// TIA Portal V17 export
// export: Created 2023-12-05T13:40:23.7935215Z, ExportSetting WithDefaults, DisplayName Totally Integrated Automation Portal, DisplayVersion V17, DisplayName TIA Portal Openness, DisplayVersion V17, DisplayName TIA Portal Version Control Interface, DisplayVersion V17, DisplayName SINAMICS Startdrive Advanced, DisplayVersion V17, DisplayName SINAMICS Startdrive G130, G150, S120, S150, SINAMICS MV, S210, DisplayVersion V17, DisplayName SINAMICS Startdrive G110M, G120, G120C, G120D, G120P, G115D, DisplayVersion V17, DisplayName STEP 7 Professional, DisplayVersion V17, DisplayName STEP 7 Safety, DisplayVersion V17, DisplayName WinCC Professional, DisplayVersion V17
FUNCTION "KNIFE_AND_SLUG_COUNTER_MANAGE" : Void   // FC402, LAD
{ S7_Optimized_Access := 'TRUE' }
VERSION : 0.1
// stored: AutoNumber false, IsIECCheckEnabled false, SetENOAutomatically false, UDAEnableTagReadback false
   VAR_TEMP   // added for the SCL form of the ladder/FBD networks
      _w1 : Bool;
      _w2 : Bool;
   END_VAR
BEGIN

REGION Network 1: -------------------------------------------------- KNIFE COUNTERS --------------------------------------------------
END_REGION

REGION Network 2: ST1OP02
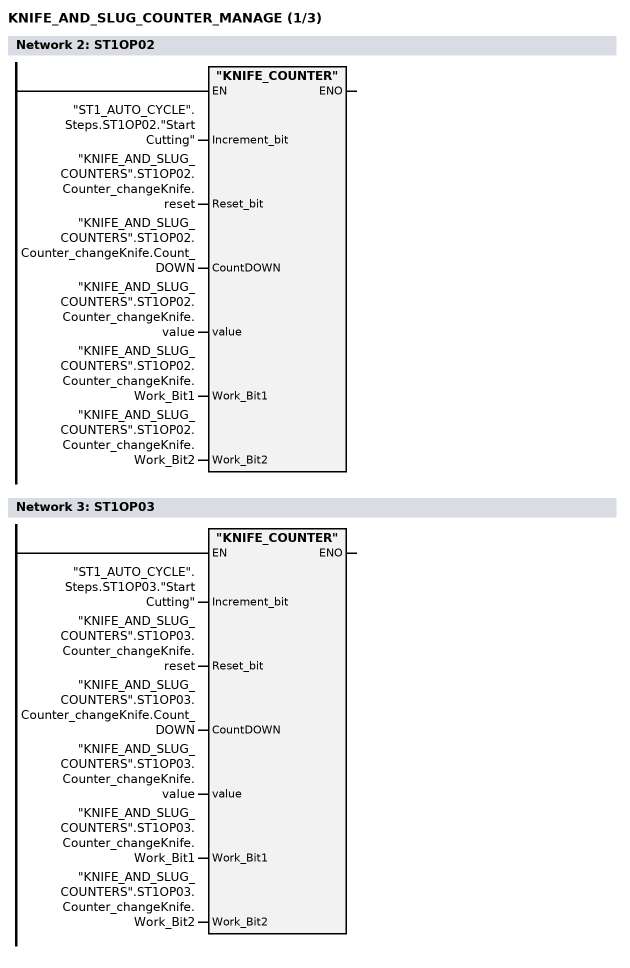
   RUNG wire#powerrail
      "KNIFE_COUNTER"(Increment_bit := "ST1_AUTO_CYCLE".Steps.ST1OP02."Start Cutting", Reset_bit := "KNIFE_AND_SLUG_COUNTERS".ST1OP02.Counter_changeKnife.reset, CountDOWN := "KNIFE_AND_SLUG_COUNTERS".ST1OP02.Counter_changeKnife.Count_DOWN, value := "KNIFE_AND_SLUG_COUNTERS".ST1OP02.Counter_changeKnife.value, Work_Bit1 := "KNIFE_AND_SLUG_COUNTERS".ST1OP02.Counter_changeKnife.Work_Bit1, Work_Bit2 := "KNIFE_AND_SLUG_COUNTERS".ST1OP02.Counter_changeKnife.Work_Bit2)
   END_RUNG
   // the same network as SCL:
   "KNIFE_COUNTER"(Increment_bit := "ST1_AUTO_CYCLE".Steps.ST1OP02."Start Cutting",
                   Reset_bit := "KNIFE_AND_SLUG_COUNTERS".ST1OP02.Counter_changeKnife.reset,
                   CountDOWN := "KNIFE_AND_SLUG_COUNTERS".ST1OP02.Counter_changeKnife.Count_DOWN,
                   value := "KNIFE_AND_SLUG_COUNTERS".ST1OP02.Counter_changeKnife.value,
                   Work_Bit1 := "KNIFE_AND_SLUG_COUNTERS".ST1OP02.Counter_changeKnife.Work_Bit1,
                   Work_Bit2 := "KNIFE_AND_SLUG_COUNTERS".ST1OP02.Counter_changeKnife.Work_Bit2);
END_REGION

REGION Network 3: ST1OP03
   RUNG wire#powerrail
      "KNIFE_COUNTER"(Increment_bit := "ST1_AUTO_CYCLE".Steps.ST1OP03."Start Cutting", Reset_bit := "KNIFE_AND_SLUG_COUNTERS".ST1OP03.Counter_changeKnife.reset, CountDOWN := "KNIFE_AND_SLUG_COUNTERS".ST1OP03.Counter_changeKnife.Count_DOWN, value := "KNIFE_AND_SLUG_COUNTERS".ST1OP03.Counter_changeKnife.value, Work_Bit1 := "KNIFE_AND_SLUG_COUNTERS".ST1OP03.Counter_changeKnife.Work_Bit1, Work_Bit2 := "KNIFE_AND_SLUG_COUNTERS".ST1OP03.Counter_changeKnife.Work_Bit2)
   END_RUNG
   // the same network as SCL:
   "KNIFE_COUNTER"(Increment_bit := "ST1_AUTO_CYCLE".Steps.ST1OP03."Start Cutting",
                   Reset_bit := "KNIFE_AND_SLUG_COUNTERS".ST1OP03.Counter_changeKnife.reset,
                   CountDOWN := "KNIFE_AND_SLUG_COUNTERS".ST1OP03.Counter_changeKnife.Count_DOWN,
                   value := "KNIFE_AND_SLUG_COUNTERS".ST1OP03.Counter_changeKnife.value,
                   Work_Bit1 := "KNIFE_AND_SLUG_COUNTERS".ST1OP03.Counter_changeKnife.Work_Bit1,
                   Work_Bit2 := "KNIFE_AND_SLUG_COUNTERS".ST1OP03.Counter_changeKnife.Work_Bit2);
END_REGION

REGION Network 4: ST2OP18
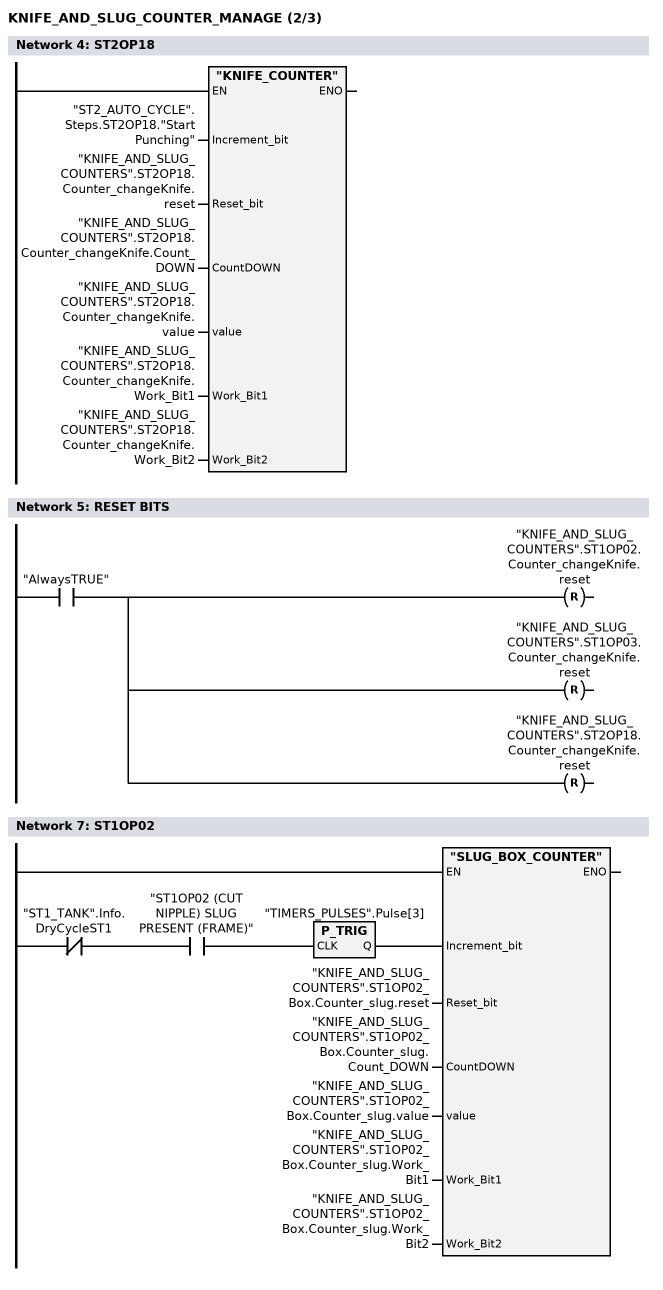
   RUNG wire#powerrail
      "KNIFE_COUNTER"(Increment_bit := "ST2_AUTO_CYCLE".Steps.ST2OP18."Start Punching", Reset_bit := "KNIFE_AND_SLUG_COUNTERS".ST2OP18.Counter_changeKnife.reset, CountDOWN := "KNIFE_AND_SLUG_COUNTERS".ST2OP18.Counter_changeKnife.Count_DOWN, value := "KNIFE_AND_SLUG_COUNTERS".ST2OP18.Counter_changeKnife.value, Work_Bit1 := "KNIFE_AND_SLUG_COUNTERS".ST2OP18.Counter_changeKnife.Work_Bit1, Work_Bit2 := "KNIFE_AND_SLUG_COUNTERS".ST2OP18.Counter_changeKnife.Work_Bit2)
   END_RUNG
   // the same network as SCL:
   "KNIFE_COUNTER"(Increment_bit := "ST2_AUTO_CYCLE".Steps.ST2OP18."Start Punching",
                   Reset_bit := "KNIFE_AND_SLUG_COUNTERS".ST2OP18.Counter_changeKnife.reset,
                   CountDOWN := "KNIFE_AND_SLUG_COUNTERS".ST2OP18.Counter_changeKnife.Count_DOWN,
                   value := "KNIFE_AND_SLUG_COUNTERS".ST2OP18.Counter_changeKnife.value,
                   Work_Bit1 := "KNIFE_AND_SLUG_COUNTERS".ST2OP18.Counter_changeKnife.Work_Bit1,
                   Work_Bit2 := "KNIFE_AND_SLUG_COUNTERS".ST2OP18.Counter_changeKnife.Work_Bit2);
END_REGION

REGION Network 5: RESET BITS
   RUNG wire#powerrail
      Contact( "AlwaysTRUE" )
      wire#w1
      R_Coil( "KNIFE_AND_SLUG_COUNTERS".ST1OP02.Counter_changeKnife.reset )
   END_RUNG
   RUNG wire#w1
      R_Coil( "KNIFE_AND_SLUG_COUNTERS".ST1OP03.Counter_changeKnife.reset )
   END_RUNG
   RUNG wire#w1
      R_Coil( "KNIFE_AND_SLUG_COUNTERS".ST2OP18.Counter_changeKnife.reset )
   END_RUNG
   // the same network as SCL:
   IF "AlwaysTRUE" THEN
       "KNIFE_AND_SLUG_COUNTERS".ST1OP02.Counter_changeKnife.reset := FALSE;
       "KNIFE_AND_SLUG_COUNTERS".ST1OP03.Counter_changeKnife.reset := FALSE;
       "KNIFE_AND_SLUG_COUNTERS".ST2OP18.Counter_changeKnife.reset := FALSE;
   END_IF;
END_REGION

REGION Network 6: -------------------------------------------------- SLUG BOX COUNTERS --------------------------------------------------
END_REGION

REGION Network 7: ST1OP02
   RUNG wire#powerrail
      "SLUG_BOX_COUNTER"(Increment_bit := wire#w1, Reset_bit := "KNIFE_AND_SLUG_COUNTERS".ST1OP02_Box.Counter_slug.reset, CountDOWN := "KNIFE_AND_SLUG_COUNTERS".ST1OP02_Box.Counter_slug.Count_DOWN, value := "KNIFE_AND_SLUG_COUNTERS".ST1OP02_Box.Counter_slug.value, Work_Bit1 := "KNIFE_AND_SLUG_COUNTERS".ST1OP02_Box.Counter_slug.Work_Bit1, Work_Bit2 := "KNIFE_AND_SLUG_COUNTERS".ST1OP02_Box.Counter_slug.Work_Bit2)
   END_RUNG
   RUNG wire#powerrail
      I_Contact( "ST1_TANK".Info.DryCycleST1 )
      Contact( "ST1OP02 (CUT NIPPLE) SLUG PRESENT (FRAME)" )
      P_Trig( "TIMERS_PULSES".Pulse[3] )
   END_RUNG wire#w1
   // the same network as SCL:
   #_w1 := NOT "ST1_TANK".Info.DryCycleST1 AND "ST1OP02 (CUT NIPPLE) SLUG PRESENT (FRAME)";
   #_w2 := #_w1 AND NOT "TIMERS_PULSES".Pulse[3];   // rising edge
   "TIMERS_PULSES".Pulse[3] := #_w1;
   "SLUG_BOX_COUNTER"(Increment_bit := #_w2,
                      Reset_bit := "KNIFE_AND_SLUG_COUNTERS".ST1OP02_Box.Counter_slug.reset,
                      CountDOWN := "KNIFE_AND_SLUG_COUNTERS".ST1OP02_Box.Counter_slug.Count_DOWN,
                      value := "KNIFE_AND_SLUG_COUNTERS".ST1OP02_Box.Counter_slug.value,
                      Work_Bit1 := "KNIFE_AND_SLUG_COUNTERS".ST1OP02_Box.Counter_slug.Work_Bit1,
                      Work_Bit2 := "KNIFE_AND_SLUG_COUNTERS".ST1OP02_Box.Counter_slug.Work_Bit2);
END_REGION

REGION Network 8: ST1OP03
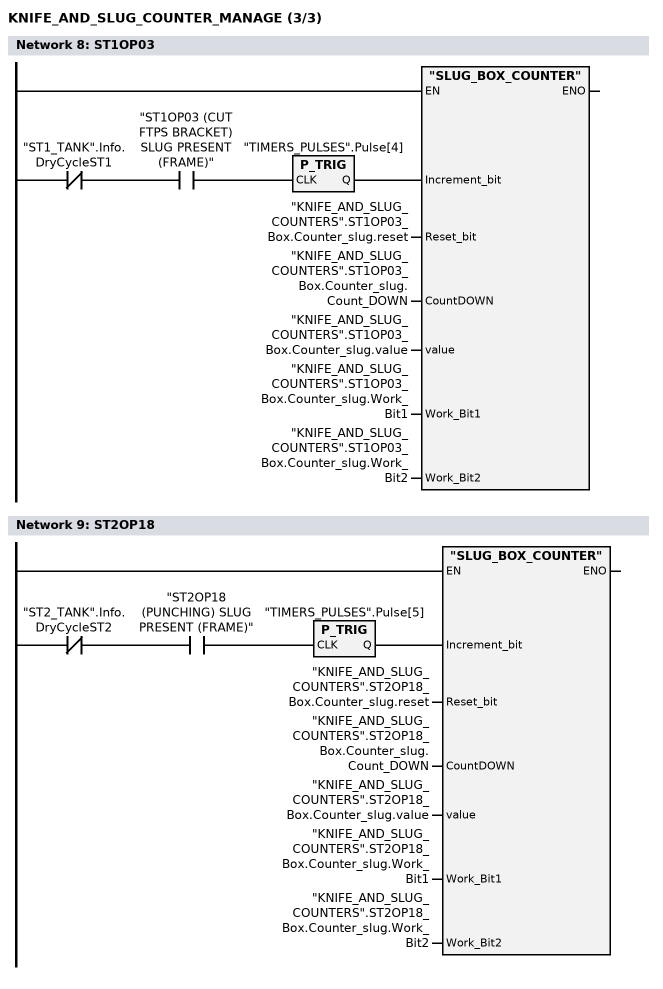
   RUNG wire#powerrail
      "SLUG_BOX_COUNTER"(Increment_bit := wire#w1, Reset_bit := "KNIFE_AND_SLUG_COUNTERS".ST1OP03_Box.Counter_slug.reset, CountDOWN := "KNIFE_AND_SLUG_COUNTERS".ST1OP03_Box.Counter_slug.Count_DOWN, value := "KNIFE_AND_SLUG_COUNTERS".ST1OP03_Box.Counter_slug.value, Work_Bit1 := "KNIFE_AND_SLUG_COUNTERS".ST1OP03_Box.Counter_slug.Work_Bit1, Work_Bit2 := "KNIFE_AND_SLUG_COUNTERS".ST1OP03_Box.Counter_slug.Work_Bit2)
   END_RUNG
   RUNG wire#powerrail
      I_Contact( "ST1_TANK".Info.DryCycleST1 )
      Contact( "ST1OP03 (CUT FTPS BRACKET) SLUG PRESENT (FRAME)" )
      P_Trig( "TIMERS_PULSES".Pulse[4] )
   END_RUNG wire#w1
   // the same network as SCL:
   #_w1 := NOT "ST1_TANK".Info.DryCycleST1 AND "ST1OP03 (CUT FTPS BRACKET) SLUG PRESENT (FRAME)";
   #_w2 := #_w1 AND NOT "TIMERS_PULSES".Pulse[4];   // rising edge
   "TIMERS_PULSES".Pulse[4] := #_w1;
   "SLUG_BOX_COUNTER"(Increment_bit := #_w2,
                      Reset_bit := "KNIFE_AND_SLUG_COUNTERS".ST1OP03_Box.Counter_slug.reset,
                      CountDOWN := "KNIFE_AND_SLUG_COUNTERS".ST1OP03_Box.Counter_slug.Count_DOWN,
                      value := "KNIFE_AND_SLUG_COUNTERS".ST1OP03_Box.Counter_slug.value,
                      Work_Bit1 := "KNIFE_AND_SLUG_COUNTERS".ST1OP03_Box.Counter_slug.Work_Bit1,
                      Work_Bit2 := "KNIFE_AND_SLUG_COUNTERS".ST1OP03_Box.Counter_slug.Work_Bit2);
END_REGION

REGION Network 9: ST2OP18
   RUNG wire#powerrail
      "SLUG_BOX_COUNTER"(Increment_bit := wire#w1, Reset_bit := "KNIFE_AND_SLUG_COUNTERS".ST2OP18_Box.Counter_slug.reset, CountDOWN := "KNIFE_AND_SLUG_COUNTERS".ST2OP18_Box.Counter_slug.Count_DOWN, value := "KNIFE_AND_SLUG_COUNTERS".ST2OP18_Box.Counter_slug.value, Work_Bit1 := "KNIFE_AND_SLUG_COUNTERS".ST2OP18_Box.Counter_slug.Work_Bit1, Work_Bit2 := "KNIFE_AND_SLUG_COUNTERS".ST2OP18_Box.Counter_slug.Work_Bit2)
   END_RUNG
   RUNG wire#powerrail
      I_Contact( "ST2_TANK".Info.DryCycleST2 )
      Contact( "ST2OP18 (PUNCHING) SLUG PRESENT (FRAME)" )
      P_Trig( "TIMERS_PULSES".Pulse[5] )
   END_RUNG wire#w1
   // the same network as SCL:
   #_w1 := NOT "ST2_TANK".Info.DryCycleST2 AND "ST2OP18 (PUNCHING) SLUG PRESENT (FRAME)";
   #_w2 := #_w1 AND NOT "TIMERS_PULSES".Pulse[5];   // rising edge
   "TIMERS_PULSES".Pulse[5] := #_w1;
   "SLUG_BOX_COUNTER"(Increment_bit := #_w2,
                      Reset_bit := "KNIFE_AND_SLUG_COUNTERS".ST2OP18_Box.Counter_slug.reset,
                      CountDOWN := "KNIFE_AND_SLUG_COUNTERS".ST2OP18_Box.Counter_slug.Count_DOWN,
                      value := "KNIFE_AND_SLUG_COUNTERS".ST2OP18_Box.Counter_slug.value,
                      Work_Bit1 := "KNIFE_AND_SLUG_COUNTERS".ST2OP18_Box.Counter_slug.Work_Bit1,
                      Work_Bit2 := "KNIFE_AND_SLUG_COUNTERS".ST2OP18_Box.Counter_slug.Work_Bit2);
END_REGION
END_FUNCTION
